INTERFACE I_AxisMoveAbsolute

(* Copy it to derived Function block if developing this function *)
PROPERTY ActualPosition : REFERENCE TO LREAL
GET
END_GET
END_PROPERTY

(* Copy it to derived Function block if developing this function *)
PROPERTY InPosition : BOOL
GET
END_GET
END_PROPERTY

METHOD MR_MoveAbsolute : BOOL
VAR_INPUT
	lrAbsolutePosition : LREAL;
END_VAR
END_METHOD

PROPERTY SetpointPosition : LREAL
GET
END_GET
END_PROPERTY

END_INTERFACE

(* stored: Version 1.1.0.1, ProductVersion 3.1.4024.12
   Itf I_AxisMoveAbsolute: Id {577851f7-436a-474f-9683-bed722c561b9}
   Property ActualPosition: Id {cf88f8da-ee83-45f7-8024-6775855e24e1}
   Get Get: Id {00301ed6-4b5c-446f-96e5-94752993dfcf}
   Property InPosition: Id {76d96262-ce60-47f5-b46a-3c38f0edb9b4}
   Get Get: Id {b146c69e-160d-4ae3-9693-96d2a8d80228}
   Method MR_MoveAbsolute: Id {4df310fb-3248-4435-be2a-9088ef3119d1}
   Property SetpointPosition: Id {2ef6fa9d-dc72-43d7-b689-e50b62128a9a}
   Get Get: Id {97ed0241-19a1-40eb-b056-34bf4c75e425} *)
